(* CoDeSys 2.3.9.50 project: 7A.pr6 *)
(* Libraries: STANDARD.LB6 5.6.98 12:03:02 *)

(* POU MAIN, LD *)
PROGRAM MAIN
VAR
	Auto AT %IX0.0: BOOL;
	manual AT %IX0.1: BOOL;
	Motor AT %QX0.0: BOOL;
	Pump AT %QX0.1: BOOL;
	Stop AT %IX0.2: BOOL;
	Start AT %IX0.3: BOOL;
	Highlevel AT %IX0.4: BOOL;
	HL AT %QX0.2: BOOL;
	LowLevel AT %IX0.5: BOOL;
	LL AT %QX0.3: BOOL;
END_VAR
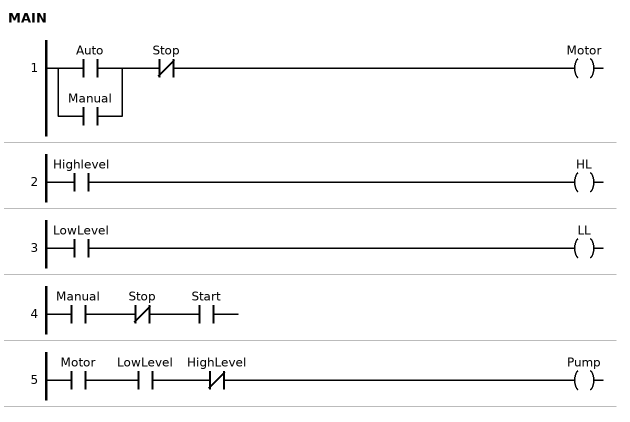
_LD_ (* Ladder Diagram *)
NETWORK 1
	{ [Auto] | [Manual] } - [/Stop] --- (Motor)
NETWORK 2
	[Highlevel] --- (HL)
NETWORK 3
	[LowLevel] --- (LL)
NETWORK 4
	[Manual] - [/Stop] - [Start]
NETWORK 5
	[Motor] - [LowLevel] - [/HighLevel] --- (Pump)
_END_LD_
(* the same logic as Structured Text *)
(* Network 1 *)
Motor := (Auto OR Manual) AND NOT Stop;
(* Network 2 *)
HL := Highlevel;
(* Network 3 *)
LL := LowLevel;
(* Network 4 *)
(* Network 5 *)
Pump := Motor AND LowLevel AND NOT HighLevel;
END_PROGRAM
